FUNCTION_BLOCK EQ_NeedleAxis (* Needle lift with down/up valves, end switches and a position sensor; equipment IO: owns its IO points, writes the output values its holder sends, reads its inputs every cycle and reports changes *)
  (* Standard: 61499-2 *)
  (* Version 0.1, 2026-09-28, Project contributors, AAU Smart Production Lab *)
  PACKAGE filler;
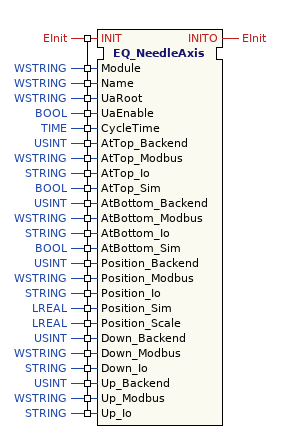
  EVENT_INPUT
    INIT : EInit WITH Module, Name, UaRoot, UaEnable, CycleTime, AtTop_Backend, AtTop_Modbus, AtTop_Io, AtTop_Sim, AtBottom_Backend, AtBottom_Modbus, AtBottom_Io, AtBottom_Sim, Position_Backend, Position_Modbus, Position_Io, Position_Sim, Position_Scale, Down_Backend, Down_Modbus, Down_Io, Up_Backend, Up_Modbus, Up_Io;
  END_EVENT
  EVENT_OUTPUT
    INITO : EInit;
  END_EVENT
  VAR_INPUT
    Module : WSTRING;
    Name : WSTRING := "NeedleAxis";
    UaRoot : WSTRING;
    UaEnable : BOOL;
    CycleTime : TIME := T#50ms;
    AtTop_Backend : USINT := 2;
    AtTop_Modbus : WSTRING;
    AtTop_Io : STRING;
    AtTop_Sim : BOOL := FALSE;
    AtBottom_Backend : USINT := 2;
    AtBottom_Modbus : WSTRING;
    AtBottom_Io : STRING;
    AtBottom_Sim : BOOL := FALSE;
    Position_Backend : USINT := 2;
    Position_Modbus : WSTRING;
    Position_Io : STRING;
    Position_Sim : LREAL := 0.0;
    Position_Scale : LREAL := 0.1;
    Down_Backend : USINT := 2;
    Down_Modbus : WSTRING;
    Down_Io : STRING;
    Up_Backend : USINT := 2;
    Up_Modbus : WSTRING;
    Up_Io : STRING;
  END_VAR
  (* Group Core: One holder at a time, break before make, all off on release or abort; scanned every CycleTime *)
  (* Group Channels: Local channels to and from the skills (cmd, release, state), the module's state, and the inputs over OPC UA *)
  (* Group Inputs: The equipment's sensors: read every cycle, one block per IO point *)
  (* Group Outputs: The equipment's actuators: written on a change and every cycle, one block per IO point *)
  FBS
    Logic : filler::EL_NeedleAxis; {SET_ATTRIBUTE(GroupName, Core)}
    Cycle : iec61499::events::E_CYCLE; {SET_ATTRIBUTE(GroupName, Core)}
    Mode : modlib::MOD_StateView; {SET_ATTRIBUTE(GroupName, Channels)}
    SubCmd : iec61499::net::SUBSCRIBE_4(QI := TRUE); {SET_ATTRIBUTE(GroupName, Channels)}
    SubRelease : iec61499::net::SUBSCRIBE_1(QI := TRUE); {SET_ATTRIBUTE(GroupName, Channels)}
    PubState : iec61499::net::PUBLISH_4(QI := TRUE); {SET_ATTRIBUTE(GroupName, Channels)}
    PubUa : iec61499::net::PUBLISH_3; {SET_ATTRIBUTE(GroupName, Channels)}
    In_AtTop : modlib::IO_DI; {SET_ATTRIBUTE(GroupName, Inputs)}
    In_AtBottom : modlib::IO_DI; {SET_ATTRIBUTE(GroupName, Inputs)}
    In_Position : modlib::IO_AI; {SET_ATTRIBUTE(GroupName, Inputs)}
    Out_Down : modlib::IO_DO; {SET_ATTRIBUTE(GroupName, Outputs)}
    Out_Up : modlib::IO_DO; {SET_ATTRIBUTE(GroupName, Outputs)}
  END_FBS
  EVENT_CONNECTIONS
    INIT TO Logic.INIT;
    Logic.INITO TO Mode.INIT;
    Mode.INITO TO SubCmd.INIT;
    SubCmd.INITO TO SubRelease.INIT;
    SubRelease.INITO TO PubState.INIT;
    PubState.INITO TO PubUa.INIT;
    PubUa.INITO TO In_AtTop.INIT;
    In_AtTop.INITO TO In_AtBottom.INIT;
    In_AtBottom.INITO TO In_Position.INIT;
    In_Position.INITO TO Out_Down.INIT;
    Out_Down.INITO TO Out_Up.INIT;
    Out_Up.INITO TO Cycle.START;
    Out_Up.INITO TO INITO;
    SubCmd.IND TO Logic.CMD;
    SubRelease.IND TO Logic.RELEASE;
    Mode.CHG TO Logic.MOD_CHG;
    Cycle.EO TO Logic.REFRESH;
    Cycle.EO TO In_AtTop.REQ;
    In_AtTop.CNF TO In_AtBottom.REQ;
    In_AtBottom.CNF TO In_Position.REQ;
    In_Position.CNF TO Logic.SAMPLE;
    Logic.STATE TO PubState.REQ;
    Logic.STATE TO PubUa.REQ;
    Logic.DRIVE TO Out_Down.REQ;
    Out_Down.CNF TO Out_Up.REQ;
    Out_Up.CNF TO Logic.DRIVEN;
  END_CONNECTIONS
  DATA_CONNECTIONS
    Module TO Logic.Module;
    Name TO Logic.Name;
    UaRoot TO Logic.UaRoot;
    Module TO Mode.Module;
    Logic.IdCmd TO SubCmd.ID;
    Logic.IdRelease TO SubRelease.ID;
    Logic.IdState TO PubState.ID;
    Logic.IdPub TO PubUa.ID;
    UaEnable TO PubUa.QI;
    CycleTime TO Cycle.DT;
    SubCmd.RD_1 TO Logic.C_Holder;
    SubCmd.RD_2 TO Logic.C_Release;
    SubCmd.RD_3 TO Logic.C_Down;
    SubCmd.RD_4 TO Logic.C_Up;
    SubRelease.RD_1 TO Logic.R_Holder;
    Mode.State TO Logic.ModState;
    AtTop_Backend TO In_AtTop.Backend;
    AtTop_Modbus TO In_AtTop.ModbusId;
    AtTop_Io TO In_AtTop.IoName;
    AtTop_Sim TO In_AtTop.SimValue;
    In_AtTop.IN TO Logic.I_AtTop;
    Logic.AtTop TO PubState.SD_1;
    Logic.AtTop TO PubUa.SD_1;
    AtBottom_Backend TO In_AtBottom.Backend;
    AtBottom_Modbus TO In_AtBottom.ModbusId;
    AtBottom_Io TO In_AtBottom.IoName;
    AtBottom_Sim TO In_AtBottom.SimValue;
    In_AtBottom.IN TO Logic.I_AtBottom;
    Logic.AtBottom TO PubState.SD_2;
    Logic.AtBottom TO PubUa.SD_2;
    Position_Backend TO In_Position.Backend;
    Position_Modbus TO In_Position.ModbusId;
    Position_Io TO In_Position.IoName;
    Position_Sim TO In_Position.SimValue;
    Position_Scale TO In_Position.Scale;
    In_Position.IN TO Logic.I_Position;
    Logic.Position TO PubState.SD_3;
    Logic.Position TO PubUa.SD_3;
    Logic.Holder TO PubState.SD_4;
    Down_Backend TO Out_Down.Backend;
    Down_Modbus TO Out_Down.ModbusId;
    Down_Io TO Out_Down.IoName;
    Logic.O_Down TO Out_Down.OUT;
    Up_Backend TO Out_Up.Backend;
    Up_Modbus TO Out_Up.ModbusId;
    Up_Io TO Out_Up.IoName;
    Logic.O_Up TO Out_Up.OUT;
  END_CONNECTIONS
END_FUNCTION_BLOCK
